// TIA Portal V16 export
// export: Created 2022-02-28T20:45:46.4622933Z, ExportSetting WithDefaults, DisplayName Totally Integrated Automation Portal, DisplayVersion V16, DisplayName TIA Portal Version Control Interface, DisplayVersion V16, DisplayName TIA Portal Openness, DisplayVersion V16, DisplayName STEP 7 Professional, DisplayVersion V16, DisplayName STEP 7 Safety, DisplayVersion V16, DisplayName WinCC Advanced, DisplayVersion V16
DATA_BLOCK "Auto-Manual Pistilos"   // DB7
VERSION : 0.1
// stored: AutoNumber true, DBAccessibleFromOPCUA true, InstanceOfName Modo_Auto-Manual, InstanceOfType FB
"Modo_Auto-Manual"
   // VAR_INPUT
   //    Confir_Perifericos : Bool;
   //    Modo_Automatico : Bool;
   //    Modo_Manual : Bool;
   //    Run_Btn : Bool;
   //    Stop_Btn : Bool;
   //    Run_HMI : Bool;
   //    Stop_HMI : Bool;
   //    Paro_Emergencia : Bool;
   //    "Remoto-Local" : Bool;
   // END_VAR
   // VAR_OUTPUT
   //    Arranque_Automatico : Bool;
   //    Arranque_Manual : Bool;
   // END_VAR
   // VAR
   //    Start_Remoto : Bool;
   //    Stop_Remoto : Bool;
   // END_VAR
BEGIN
END_DATA_BLOCK
